FUNCTION_BLOCK RangeSensor (* Basic Function Block Type *)
  (* Standard: 61499-2 *)
  (* Version 0.0, 12/5/2011, XPMUser, nxtControl GmbH, Template *)
  PACKAGE Main;
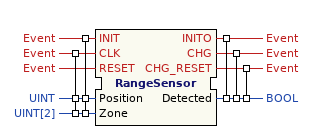
  EVENT_INPUT
    INIT WITH Position, Zone; (* Initialization Request *)
    CLK WITH Position, Zone; (* Clock signal *)
    RESET;
  END_EVENT
  EVENT_OUTPUT
    INITO WITH Detected; (* Initialization Confirm *)
    CHG WITH Detected; (* Value of DETECTED changed *)
    CHG_RESET WITH Detected;
  END_EVENT
  VAR_INPUT
    Position : UINT; (* The object's position *)
    Zone : ARRAY [0..1] OF UINT; (* Detection range of the sensor *)
  END_VAR
  VAR_OUTPUT
    Detected : BOOL; (* Whether an object is detected *)
  END_VAR
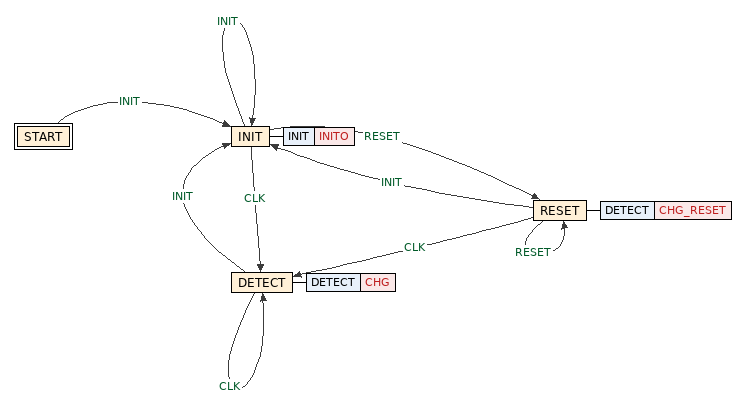
  EC_STATES
    START; (* Initial State *)
    INIT : INIT -> INITO; (* Initialization *)
    DETECT : DETECT -> CHG; (* Detect *)
    RESET : DETECT -> CHG_RESET;
  END_STATES
  EC_TRANSITIONS
    START TO INIT := INIT;
    INIT TO DETECT := CLK;
    DETECT TO DETECT := CLK;
    DETECT TO INIT := INIT;
    INIT TO INIT := INIT;
    INIT TO RESET := RESET;
    RESET TO DETECT := CLK;
    RESET TO RESET := RESET;
    RESET TO INIT := INIT;
  END_TRANSITIONS
  ALGORITHM INIT IN ST: (* Initialization algorithm *)
INIT:=FALSE;
IF ((Position >= Zone[0]) AND ( Position <= Zone[1])) THEN
  Detected := TRUE;
ELSE
  Detected := FALSE;
END_IF;
  END_ALGORITHM
  ALGORITHM DETECT IN ST: (* Normally executed algorithm *)
RESET:=FALSE;
IF ((Position >= Zone[0]) AND ( Position <= Zone[1])) THEN
  IF (Detected = FALSE) THEN
      Detected := TRUE;
      (*CHG := CHG+1;*)
  END_IF;
ELSE
  IF (Detected = TRUE) THEN
      Detected := FALSE;
      (*CHG := CHG+1;*)
  END_IF;
END_IF;
  END_ALGORITHM
END_FUNCTION_BLOCK
